Staubli VAL3: JointFbkMsg.pjx

--- JointFbkMsg.pjx ---
Parameters version=s7.7.2 stackSize=5000 millimeterUnit=true
Program file=start.pgx
Program file=stop.pgx
Data file=JointFbkMsg.dtx
Type name=Body path=Disk://ros_libs/Body/Body.pjx
Type name=Header path=Disk://ros_libs/Header/Header.pjx
Type name=Prefix path=Disk://ros_libs/Prefix/Prefix.pjx
Type name=JointFeedback path=Disk://ros_libs/JointFeedback/JointFeedback.pjx

--- JointFbkMsg.dtx ---
public Header header
  [0]
    num nMsgType
    num nCommType
    num nReplyCode
    num nData[12]
public Prefix prefix
  [0]
    num nLength
    num nData[4]
public JointFeedback jointFeedback
  [0]
    num nRobotId
    num nValidFields
    num nTime
    num nPositions[10]
    num nVelocities[10]
    num nAccelerations[10]
public Body body
  [0]
    num nData[132]
